FUNCTION_BLOCK State_Levi_Testing_Individual_Drives
VAR_INPUT
	drive_status: ARRAY [0..23] OF UINT;
	drive_diagnostics: ARRAY [0..23] OF UINT;
	State : E_Levi_States;
	Force_feedback_value : ARRAY[0..23] OF INT;
END_VAR

VAR_OUTPUT
	Error: BOOL;
	Run_z_liftoff_calc : BOOL;
END_VAR

VAR_IN_OUT
	Control_word_array : ARRAY[0..23] OF UINT;
	drive_feedback_timeouts : ARRAY[0..23] OF UINT;
	force_values : ARRAY[0..11] OF INT;
	Drive_current_error : ARRAY[0..23] OF BOOL;
	error_specifics: ARRAY [0..23] OF Drive_error_mapping;
END_VAR

VAR
	count_cycles: INT;
	n_drive_warnings: UINT;
	n_drive_errors: UINT;
	
	Control_word_VFL1_N : UINT;
	Control_word_VFL1_S : UINT;
	Control_word_VFL2_N : UINT;
	Control_word_VFL2_S : UINT;
	Control_word_VFR1_N : UINT;
	Control_word_VFR1_S : UINT;
	Control_word_VFR2_N : UINT;
	Control_word_VFR2_S : UINT;
	Control_word_VBL1_N : UINT;
	Control_word_VBL1_S : UINT;
	Control_word_VBL2_N : UINT;
	Control_word_VBL2_S : UINT;
	Control_word_VBR1_N : UINT;
	Control_word_VBR1_S : UINT;
	Control_word_VBR2_N : UINT;
	Control_word_VBR2_S : UINT;
	Control_word_LF1_N : UINT;
	Control_word_LF1_S : UINT;
	Control_word_LF2_N : UINT;
	Control_word_LF2_S : UINT;
	Control_word_LB1_N : UINT;
	Control_word_LB1_S : UINT;
	Control_word_LB2_N : UINT;
	Control_word_LB2_S : UINT;
	
	TestVFL1 : LREAL;
	TestVFL2 : LREAL;
	TestVFR1 : LREAL;
	TestVFR2 : LREAL;
	TestVBL1 : LREAL;
	TestVBL2 : LREAL;	
	TestVBR1 : LREAL;	
	TestVBR2: LREAL;
	TestLF1 : LREAL;
	TestLF2 : LREAL;
	TestLB1 : LREAL;
	TestLB2 : LREAL;
	
	Switch_on_individual_test : BOOL;
	
	i: INT;
END_VAR

Control_word_array[0] := Control_word_VFL1_N;
Control_word_array[1] := Control_word_VFL1_S;
Control_word_array[2] := Control_word_VFL2_N;
Control_word_array[3] := Control_word_VFL2_S;
Control_word_array[4] := Control_word_VFR1_N;
Control_word_array[5] := Control_word_VFR1_S;
Control_word_array[6] := Control_word_VFR2_N;
Run_z_liftoff_calc := FALSE;

Control_word_array[7] := Control_word_VFR2_S;
Control_word_array[8] := Control_word_VBL1_N;
Control_word_array[9] := Control_word_VBL1_S;
Control_word_array[10] := Control_word_VBL2_N;
Control_word_array[11] := Control_word_VBL2_S;
Control_word_array[12] := Control_word_VBR1_N;
Control_word_array[13] := Control_word_VBR1_S;
Control_word_array[14] := Control_word_VBR2_N;
Control_word_array[15] := Control_word_VBR2_S;

Control_word_array[16] := Control_word_LF1_N;
Control_word_array[17] := Control_word_LF1_S;
Control_word_array[18] := Control_word_LF2_N;
Control_word_array[19] := Control_word_LF2_S;
Control_word_array[20] := Control_word_LB1_N;
Control_word_array[21] := Control_word_LB1_S;
Control_word_array[22] := Control_word_LB2_N;
Control_word_array[23] := Control_word_LB2_S;

(*
GVL_LEVI.Control_lat_parameters.blevi_operational := FALSE;
GVL_LEVI.Control_vert_parameters.blevi_operational := FALSE;
GVL_LEVI.FB_Control_lat.stlateral_levitation_control_P := GVL_LEVI.Control_lat_parameters;
GVL_LEVI.FB_Control_vert.stvertical_levitation_control_P := GVL_LEVI.Control_vert_parameters;
*)

//Check if there are errors
Error := Check_drives(drive_status := drive_status, 
					drive_diagnostics := drive_diagnostics, 
					drive_last_request_value := force_values,
					drive_last_feedback_value := Force_feedback_value,
					drive_feedback_timeouts := drive_feedback_timeouts,
					State := State,
					errors := error_specifics,
					Drive_current_error := Drive_current_error,
					n_warns => n_drive_warnings, 
					n_errors => n_drive_errors);

IF Switch_on_individual_test = TRUE THEN

	force_values[0] := LREAL_TO_INT((TestVFL1 * 1000.0)/ GVL_LEVI.configured_peak_current_hems);
	force_values[1] := LREAL_TO_INT((TestVFL2 * 1000.0)/ GVL_LEVI.configured_peak_current_hems);
	
	force_values[2] := LREAL_TO_INT((TestVFR1 * 1000.0)/ GVL_LEVI.configured_peak_current_hems);
	force_values[3] := LREAL_TO_INT((TestVFR2 * 1000.0)/ GVL_LEVI.configured_peak_current_hems);
	
	force_values[4] := LREAL_TO_INT((TestVBL1 * 1000.0)/ GVL_LEVI.configured_peak_current_hems);
	force_values[5] := LREAL_TO_INT((TestVBL2 * 1000.0)/ GVL_LEVI.configured_peak_current_hems);
	
	force_values[6] := LREAL_TO_INT((TestVBR1 * 1000.0)/ GVL_LEVI.configured_peak_current_hems);
	force_values[7] := LREAL_TO_INT((TestVBR2 * 1000.0)/ GVL_LEVI.configured_peak_current_hems);
	
	force_values[8] := LREAL_TO_INT((TestLF1 * 1000.0)/ GVL_LEVI.configured_peak_current_ems);
	force_values[9] := LREAL_TO_INT((TestLF2 * 1000.0)/ GVL_LEVI.configured_peak_current_ems);
	
	force_values[10] := LREAL_TO_INT((TestLB1 * 1000.0)/ GVL_LEVI.configured_peak_current_ems);
	force_values[11] := LREAL_TO_INT((TestLB2 * 1000.0)/ GVL_LEVI.configured_peak_current_ems);
	
ELSIF Switch_on_individual_test = FALSE THEN
	
	force_values[0] := 0;
	force_values[1] := 0;
	
	force_values[2] := 0;
	force_values[3] := 0;
	
	force_values[4] := 0;
	force_values[5] := 0;
	
	force_values[6] := 0;
	force_values[7] := 0;
	
	force_values[8] := 0;
	force_values[9] := 0;
	
	force_values[10] := 0;
	force_values[11] := 0;

END_IF

END_FUNCTION_BLOCK

(* stored: Version 1.1.0.1
   POU State_Levi_Testing_Individual_Drives: Id {ac532a27-55be-4c53-8776-155af2a2c6e5}, SpecialFunc None *)
